{attribute 'qualified_only'}
VAR_GLOBAL 
	//for downstream
	//downstreamSyncEngaged AT%MB127 : BOOL;
	//downstreamSyncAcknowledged AT%MB128 : BOOL;

	//
	//fakeInput AT%I* : bool;
	
	materialSlots : ARRAY[1..3] OF Block128Words;	
	axisControls: ARRAY[1..8] OF RunAxis;
	stations : ARRAY[1..32] OF POINTER TO RunUnitGeneric;
	
	cylinderControls : ARRAY[1..32] OF RunCylinder;
	signalControls : ARRAY[1..16] OF RunSignal;
	
END_VAR
VAR_GLOBAL RETAIN
	//commandBlocks : ARRAY[1..128] OF ParameterSet;
	bObjectsLinked : BOOL;
END_VAR

(* stored: Version 1.1.0.1, ProductVersion 3.1.4022.10
   GVL GVL: Id {e607aa11-c301-416f-9cbc-bc4f43af5299} *)
